PROGRAM RunTests
VAR
    fbAtomicMass_Test : FB_AtomicMass_Test;
    fbAtomicNumber_Test : FB_AtomicNumber_Test;
    fbElementDensity_Test : FB_ElementDensity_Test;
    fbf1Chantler_Test : FB_f1Chantler_Test;
    fbScatteringFactorLUT_Test : FB_ScatteringFactorLUT_Test;
    fbTransmission_Test : FB_Transmission_Test;

    fbCalcFocalLengthLensSet_Test : FB_CalcFocalLengthLensSet_Test;
    fbCalcFocalLengthSingleLens_Test : FB_CalcFocalLengthSingleLens_Test;
    fbCalcImageDistance_Test : FB_CalcImageDistance_Test;
    fbCalcXRayDeltaElement_Test : FB_CalcXRayDeltaElement_Test;
    fbLagrangePolyInterp_Test : FB_LagrangePolyInterp_Test;
    fbLensCompounder_Test : FB_LensCompounder_Test;

    (* Smoke test - just instantiate *)
    fbPhysicalConstants : FB_PhysicalConstants;
END_VAR


TcUnit.RUN();

fbPhysicalConstants();

END_PROGRAM

(* stored: Version 1.1.0.1
   POU RunTests: Id {3c99bab2-48fb-4f3c-ae2b-1547c32b95ba}, SpecialFunc None *)
